{attribute 'qualified_only'}
{attribute 'strict'}
{attribute 'to_string'}
TYPE EnvironmentStateEnum :
(
ready	:=	0	,//	The SystemEnvironment is in ready-state.
error	:=	100	//	The SystemEnvironment is in error.



);
END_TYPE

(* stored: Version 1.1.0.1, ProductVersion 3.1.4024.11
   DUT EnvironmentStateEnum: Id {a2e71e64-3682-4d36-8c9c-a894b73854cd} *)
